FUNCTION_BLOCK Sensors
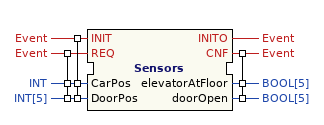
  EVENT_INPUT
    INIT WITH CarPos, DoorPos;
    REQ WITH CarPos, DoorPos;
  END_EVENT
  EVENT_OUTPUT
    INITO;
    CNF WITH elevatorAtFloor, doorOpen;
  END_EVENT
  VAR_INPUT
    CarPos : INT;
    DoorPos : ARRAY [0..4] OF INT;
  END_VAR
  VAR_OUTPUT
    elevatorAtFloor : ARRAY [0..4] OF BOOL;
    doorOpen : ARRAY [0..4] OF BOOL;
  END_VAR
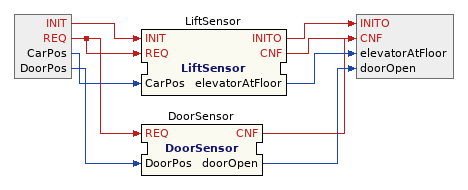
  FBS
    LiftSensor : LiftSensor;
    DoorSensor : DoorSensor;
  END_FBS
  EVENT_CONNECTIONS
    REQ TO LiftSensor.REQ;
    LiftSensor.CNF TO CNF;
    REQ TO DoorSensor.REQ;
    DoorSensor.CNF TO CNF;
    INIT TO LiftSensor.INIT;
    LiftSensor.INITO TO INITO;
  END_CONNECTIONS
  DATA_CONNECTIONS
    CarPos TO LiftSensor.CarPos;
    DoorPos TO DoorSensor.DoorPos;
    DoorSensor.doorOpen TO doorOpen;
    LiftSensor.elevatorAtFloor TO elevatorAtFloor;
  END_CONNECTIONS
END_FUNCTION_BLOCK
